// Mitsubishi GX Works2 project: fb_test   PLC: Q03UDV

// task Task_01 (event TRUE, interval 0, priority 31): MAIN

PROGRAM MAIN
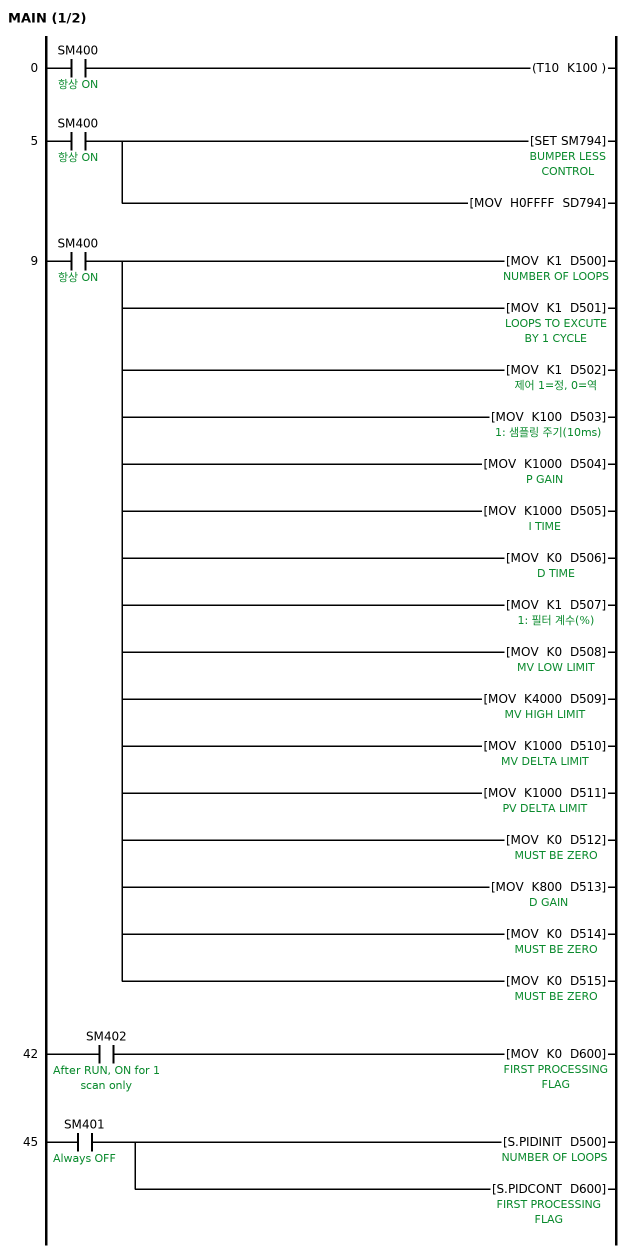
0     LD      SM400  ; 항상 ON
      OUT     T10 K100
5     LD      SM400  ; 항상 ON
      SET     SM794  ; BUMPER LESS CONTROL
      MOV     H0FFFF SD794
9     LD      SM400  ; 항상 ON
      MOV     K1 D500  ; NUMBER OF LOOPS
      MOV     K1 D501  ; LOOPS TO EXCUTE BY 1 CYCLE
      MOV     K1 D502  ; 제어 1=정, 0=역
      MOV     K100 D503  ; 1: 샘플링 주기(10ms)
      MOV     K1000 D504  ; P GAIN
      MOV     K1000 D505  ; I TIME
      MOV     K0 D506  ; D TIME
      MOV     K1 D507  ; 1: 필터 계수(%)
      MOV     K0 D508  ; MV LOW LIMIT
      MOV     K4000 D509  ; MV HIGH LIMIT
      MOV     K1000 D510  ; MV DELTA LIMIT
      MOV     K1000 D511  ; PV DELTA LIMIT
      MOV     K0 D512  ; MUST BE ZERO
      MOV     K800 D513  ; D GAIN
      MOV     K0 D514  ; MUST BE ZERO
      MOV     K0 D515  ; MUST BE ZERO
42    LD      SM402  ; After RUN, ON for 1 scan only
      MOV     K0 D600  ; FIRST PROCESSING FLAG
45    LD      SM401  ; Always OFF
      S.PIDINIT D500
      S.PIDCONT D600
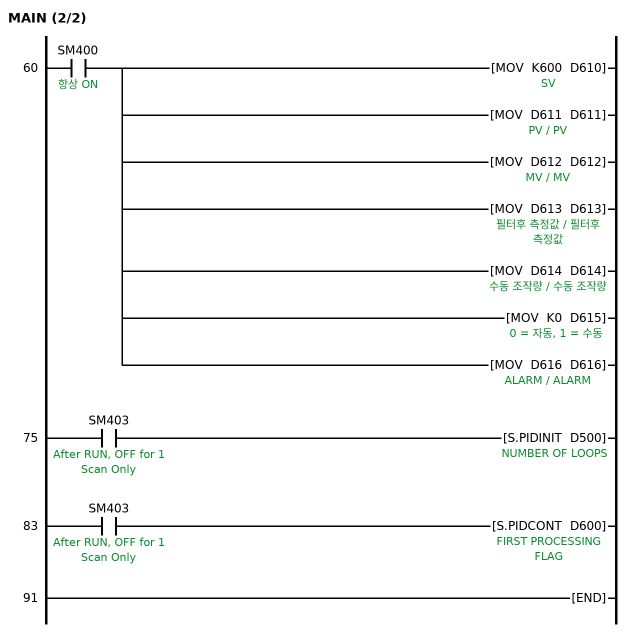
60    LD      SM400  ; 항상 ON
      MOV     K600 D610  ; SV
      MOV     D611 D611  ; PV
      MOV     D612 D612  ; MV
      MOV     D613 D613  ; 필터후 측정값
      MOV     D614 D614  ; 수동 조작량
      MOV     K0 D615  ; 0 = 자동, 1 = 수동
      MOV     D616 D616  ; ALARM
75    LD      SM403  ; After RUN, OFF for 1 Scan Only
      S.PIDINIT D500
83    LD      SM403  ; After RUN, OFF for 1 Scan Only
      S.PIDCONT D600
91    END
END_PROGRAM

// device comments not shown above
D516  ; 1=REV ACT, 0 = NOR ACT
D517  ; SAMPING TIME [10ms]
D518  ; P GAIN
D519  ; I TIME
D520  ; D TIME
D521  ; FILTER
D522  ; MV LOW LIMIT
D523  ; MV HIGH LIMIT
D524  ; MV DELTA LIMIT
D525  ; PV DELTA LIMIT
D527  ; D GAIN
